// TIA Portal V20 export
TYPE "LKinCtrl_typeJogFrameDiagnostics"
// support: tech.team.motioncontrol@siemens.com
   STRUCT
      timeStamp : Date_And_Time;   // Time stamp at which the error occurred
      status : Word;   // Status of FB when error occurred
      stateNumber : DInt;   // State in the state machine of the FB when the error occurred
   END_STRUCT;
END_TYPE
